PROGRAM MAIN 
VAR 
	fbMotorJog			:	FB_MotorJog;
	fbCamera			:	FB_Camera;
	fbMagStirrer		:	FB_MagStirrer;
// 	fbQRcode			:	FB_Camera;
// 	fbTest 				: FB_Test;
	fbEL6001	: FB_SerialCom;
	
	plcIN0 AT%I* : ARRAY [0..7] OF UINT;	//inputs w.r.t. PLC
	plcIN1 AT%I* : ARRAY [0..7] OF UINT;
	plcIN2 AT%I* : ARRAY [0..7] OF UINT;
	plcIN3 AT%I* : ARRAY [0..7] OF UINT;

	plcOUT1 AT%Q* : ARRAY [0..7] OF UINT;	//outputs w.r.t. PLC
	plcOUT2 AT%Q* : ARRAY [0..7] OF UINT;
	plcOUT3 AT%Q* : ARRAY [0..7] OF UINT;	
	plcOUT0 AT%Q* : ARRAY [0..7] OF UINT;	
	bIndex				:	USINT	:=2;
	fSuccess: BOOL;
	
END_VAR

// fbTest();
fbCamera.TriggerCamera();
// fbMotorJog.CapContainer();
// fSuccess := fbSoftwareTrigger.DetectQRCode();
fbEL6001(TxBuffer:=process_gvl.TxBufferEL, RxBuffer:=process_gvl.RxBufferEL);

	plcIN1[0].0;		// DO209	
	plcOUT1[0].0;		// DI209
	plcOUT1[0].1;		// DI210
	plcOUT1[0].2;		// DI211
	

// hr := F_VN_ReadQRCodeExp(ipImageIn, ipDecodedData, ipContours, nCodeNumber,
// 		 eSearchStrategy, hr);
// 		 
// hr := F_VN_DrawContours(ipCodeContourList, 0, ipImageRes, aColorRed, 3, hr);

END_PROGRAM

(* stored: Version 1.1.0.1
   POU MAIN: Id {5ffd7926-5d16-4ef4-80ac-73e67cfe458d}, SpecialFunc None *)
